Fanuc KAREL source: IO0219.KL

-- PROVISIONAL review KL for V1013-1; original PC SHA256 0cc6bb35e50e1c6aeb648b14822cb1cb31f1dff87a94bed075d3263a371d1405
-- Incomplete behavior may be omitted. Consult companion uncertainty JSON. Do not deploy.
PROGRAM IO0219
%NOLOCKGROUP
-- UNRESOLVED_LOCAL_POOL 5 cells at code offset 13; source declarations unknown
-- DIRECT_LOCAL_WORD_ACCESS alone does not prove INTEGER, REAL, or BOOLEAN
BEGIN
  -- UNRESOLVED_PC offsets 0-18; opcodes 2B,2C,7B
  -- UNRESOLVED_PC offsets 23-30; opcodes 9D,23
  -- UNRESOLVED_PC offsets 35-49; opcodes 2E,22,9D,33,35
  -- UNRESOLVED_PC offsets 54-61; opcodes 9D,23
  -- UNRESOLVED_PC offsets 66-77; opcodes 2E,23
  -- UNRESOLVED_PC offsets 82-103; opcodes 22,9D,33,32,36,4A
  -- UNRESOLVED_PC offsets 108-112; opcodes 7F
  -- UNRESOLVED_PC offsets 117-121; opcodes 27,AA
  -- UNRESOLVED_PC offsets 126-130; opcodes 7F
END IO0219
